(* IEC 61131-3 sources: Everest-Indoor-Unit/SWNOVHIDUOUCR00/SWNOVHIDUOUCR00/Sources/Functions/Utils, 6 files *)

(* ---- GetPasseParToutPwd.st ---- *)
FUNCTION GetPasseParToutPwd : UINT
	USING System.Timer;

    VAR
		Date : DateTime;
	END_VAR

	GetLocalTime(Date);
    GetPasseParToutPwd := 9999 - ((Date.Day * Date.Month) + Date.Year);
END_FUNCTION

(* ---- SplitString.st ---- *)
(**Split the given string in multiple rows*)
FUNCTION SplitString
	USING System;
	USING System.Text;

    VAR_INPUT
        Str : STRING;
		MaxStrLength : UDINT;
    END_VAR
	VAR_IN_OUT
	    StrArr : ARRAY[*] OF STRING;
	END_VAR
	VAR
	    i : UDINT;
		j : DINT;
		idx : DINT;
		TmpStr : STRING;
		StrLen : UDINT;
	END_VAR

	//Start index from the lower array index
	idx := LOWER_BOUND(StrArr, 1);

	StrLen := TO_UDINT(LEN(Str));

	WHILE i < StrLen DO
		//Avoid array out of bound
		IF idx > UPPER_BOUND(StrArr, 1) THEN
			EXIT;
		END_IF;

		//Pick 22 character from the string
		TmpStr := MID(Str, MaxStrLength, i + 1);

		//Check if the partial string starts with whitespace, if yes remove it.
		IF LEFT(TmpStr, 1) = ' ' THEN
			i := i + 1;
		    //Pick the new 22 character from the string
			TmpStr := MID(Str, MaxStrLength, i + 1);
		END_IF;

		(*
		1. Be sure we are NOT splitting the last 22 chars of the string otherwise it could split these chars in more lines...
		2. Check if the partial string is ending with a word
		*)
		IF i + MaxStrLength < StrLen AND MID(Str, 1, i + MaxStrLength + 1) <> ' ' THEN
		    //Find the latest word, we don't want to split the word in more lines
			FOR j := TO_DINT(MaxStrLength) TO 1 BY -1 DO
			    IF MID(TmpStr, 1, j) = ' ' THEN
					TmpStr := LEFT(TmpStr, j);
					EXIT;
				END_IF;
			END_FOR;

			//If "j" is 0 it means that the string is a long word, so the next iteration needs to increase by 22
			IF j = 0 THEN
				j := TO_DINT(MaxStrLength);
			END_IF;
		ELSE
			j := TO_DINT(MaxStrLength);
		END_IF;
		StrArr[idx] := TmpStr;
		i := i + TO_UDINT(j);
		idx := idx + 1;
	END_WHILE;
END_FUNCTION

(* ---- TruncRealString.st ---- *)
USING System;
USING System.Math;
USING System.Text;

FUNCTION truncRealString : STRING

    VAR_INPUT
        string : STRING;
        precision : DINT;
    END_VAR
    IF precision <= 0 THEN
        precision := - 1;
    END_IF;

    truncRealString := LEFT(string, FIND(string, '.') + precision);
    truncRealString := truncRealString;
END_FUNCTION

(* ---- uValueToInt.st ---- *)
USING System;

FUNCTION uValueToInt : INT

    VAR_INPUT
        value : uValue;
        dataType : DataType;
    END_VAR

    // Note: if a datatype not present below is needed, it's enough to add a new case with the proper conversion to string
    CASE dataType OF
        DataType#BOOL   : uValueToInt := TO_INT(value.bool);
        DataType#SINT   : uValueToInt := TO_INT(value.sint);
        DataType#USINT  : uValueToInt := TO_INT(value.usint);
        DataType#INT    : uValueToInt := TO_INT(value.int);
        DataType#UINT   : uValueToInt := TO_INT(value.uint);
        DataType#DINT   : uValueToInt := TO_INT(value.dint);
        DataType#UDINT  : uValueToInt := TO_INT(value.udint);
        DataType#LINT   : uValueToInt := TO_INT(value.lint);
        DataType#ULINT  : uValueToInt := TO_INT(value.ulint);
        DataType#REAL   : uValueToInt := TO_INT(value.real);
    ELSE
        uValueToInt := -999;
    END_CASE;
END_FUNCTION

(* ---- uValueToString.st ---- *)
USING System;
USING System.Math;

FUNCTION uValueToString : STRING

    VAR_INPUT
        value       : uValue;
        dataType    : DataType;
        precision   : DINT;
    END_VAR

    // Note: if a datatype not present below is needed, it's enough to add a new case with the proper conversion to string
    CASE dataType OF
        DataType#BOOL   : uValueToString := SEL(value.bool, 'FALSE', 'TRUE');
        DataType#SINT   : uValueToString := TO_STRING(value.sint);
        DataType#USINT  : uValueToString := TO_STRING(value.usint);
        DataType#INT    : uValueToString := TO_STRING(value.int);
        DataType#UINT   : uValueToString := TO_STRING(value.uint);
        DataType#DINT   : uValueToString := TO_STRING(value.dint);
        DataType#UDINT  : uValueToString := TO_STRING(value.udint);
        DataType#LINT   : uValueToString := TO_STRING(value.lint);
        DataType#ULINT  : uValueToString := TO_STRING(value.ulint);
        DataType#BYTE   : uValueToString := TO_STRING(value.byte);
        DataType#WORD   : uValueToString := TO_STRING(value.word);
        DataType#DWORD  : uValueToString := TO_STRING(value.dword);
        DataType#LWORD  : uValueToString := TO_STRING(value.lword);
        DataType#REAL   : uValueToString := truncRealString(TO_STRING(value.real), precision);
        DataType#STRING : uValueToString := value.string;
    ELSE
        uValueToString  := 'UNDEFINED';
    END_CASE;

END_FUNCTION

(* ---- DigitConv.st ---- *)
USING System;
USING System.Timer;
USING System.Math;

FUNCTION_BLOCK DigitConv
    VAR_INPUT
        Input : INT;
    END_VAR
    VAR_OUTPUT

        Digit_0   : INT;
        Digit_1   : INT;
        Digit_2   : INT;
        Digit_3   : INT;
        Digit_4   : INT;
        Digit_Sign: BOOL;

    END_VAR

    VAR
        Input_Int : INT;
    END_VAR

    IF Input<=-1 THEN
	    Digit_Sign:=TRUE;
	    Input_Int:=(-1*Input);
    ELSE
	    Digit_Sign:=FALSE;
	    Input_Int:=(Input);
    END_IF;

    Digit_4:=Input_Int/10000;
    Digit_3:=(Input_Int-Digit_4*10000)/1000;
    Digit_2:=(Input_Int-Digit_4*10000-Digit_3*1000)/100;
    Digit_1:=(Input_Int-Digit_4*10000-Digit_3*1000-Digit_2*100)/10;
    Digit_0:=(Input_Int-Digit_4*10000-Digit_3*1000-Digit_2*100-Digit_1*10)/1;
END_FUNCTION_BLOCK
